// TIA Portal V19 export
FUNCTION_BLOCK "LAF_MemCardDiag"   // FB59, LAD
TITLE = LAF_MemCardDiag / SiemensMemoryCard Diagnose mit ProDiag
AUTHOR : Siemens Digital Industries
FAMILY : LAF
VERSION : 1.2
// Information about the inserted SIMATIC memory card are retrieved, such as  
// * Memory size and assigned memory space of the memory card.  
// * Previously used up portion of the service life (lifetime) and set proportion of the lifetime of the memory card.  
// The data is evaluated in the FB, incl. ProDiag supervisions; it is displayed on the HMI in screen "Settings - PLC & HMI".
// 
// **PLC-Data types**  
// * LAF_typeMemCardDiag  
// * LAF_typeMemCardMessages  
// 
// 
// **WinCC-Screen**  
// 
// ![Image](LAF_MemCardDiag_PrD/en/image2.PNG)
//  
// **Block call example**  
// {.pageWidth}
// ![Image](LAF_MemCardDiag_PrD/en/image10.PNG)
// View in ladder logic (LAD).  
// 
// **Calling interface**  
// The block will be called once only in the cyclic program. The call takes place in the software unit CentralFunctions -> 05_Diagnostic -> [CallDiagnostic](../Functions/CallDiagnostic.htm)  
//   
// 
// **Internally used “Extended instructions / blocks”**  
// GetSMCinfo  
// 
// **Parameters**  
// 
// This block is provided with “pre-defined actual parameters” for structured data types, user constants, system constants etc. Therefor these parameters have to be modified only slightly or not at all, if the symbols of DBs, user constants, and system constants have not been changed.
// Es werden Informationen über die in der CPU gesteckte Memory Card ausgelesen, wie:  
// * Zur Verfügung stehender und benutzter Speicherplatz der Memory Card 
// * Verbrauchter Anteil und Parametrierter Anteil der Lebensdauer der Memory Card 
// 
// Die Daten werden in dem FB ausgewertet incl. ProDiag-Meldungen und auf dem HMI im Bild „SYSTEM_SETTINGS“ und im Bildbaustein „SMC_Diag“ dargestellt.  
// * LSicar_MemCardDiag_PrD:		mit ProDiag-Meldeverfahren 
// * LSicar_MemCardDiag		mit program_Alarm Meldeverfahren 
// 
// **PLC-Datentypen**  
// * LSicar_typeMemCardDiag 
// * LSicar_typeMemCardMessages  
// 
// 
// **WinCC-Faceplate**  
// 
// ![Image](LSicar_MemCardDiag_PrD/de/image1.PNG)
// 
// **WinCC-Bild**  
// 
// ![Image](LSicar_MemCardDiag_PrD/de/image2.PNG)
//  
// **Beispielaufruf**  
// Abbildung in Kontaktplan (KOP), ohne Parameterbeschaltung.  
// 
// **Aufrufschnittstelle**  
// Der Baustein wird einmalig im zyklischen Programm aufgerufen im FC „CallDiagnostic“  
// 
// **Intern verwendete „Erweiterte Anweisungen / Instructions“**  
// GetSMCinfo  
// 
// **Parameter**  
// 
// ![Icon](_Icon/information.PNG)
// 
// Der Baustein ist mit "Vordefinierten Aktualparametern" versehen für Strukturvariablen, Anwender- und Systemkonstanten etc., die dadurch nicht oder nur geringfügig angepasst werden müssen, vorausgesetzt die Symbolischen Namen von DBs, Anwender-/Systemkonstanten etc. wurden nicht geändert. Die Anpassungen sind notwendig beim Index [i], z.B. für den BA-Bereich oder die HMI-/Panelnummer.  
// * Der Index ist vorbesetzt mit dem Wert [0]. Damit wird auf den Index 0 (Dummy) verwiesen. Sofern der Baustein-Parameter nicht benötigt wird, sind keine Anpassungen notwendig, andernfalls muss der Indexwert angepasst werden. 
// oder  
// * Der Index ist vorbesetzt mit [???]. Dies führt dazu, dass der Aktualparameter beim Bausteinaufruf rot markiert wird; um darauf aufmerksam zu machen, dass der Indexwert des Aktualparameters angepasst werden muss!
// stored: Access Published, IsIECCheckEnabled true, MemoryReserve 100, SetENOAutomatically true
   VAR_INPUT
      plantIdentifier { ExternalAccessible := 'False'; ExternalVisible := 'False'; ExternalWritable := 'False'} : WString[#MAX_CHAR];   // Betriebsmittel Kennzeichen. Das Kennzeichen ist auf 24 Zeichen begrenzt und sollte ein Betriebsmittelkennzeichen, gemäß der Schaltpläne enthalten. Der hier angegebene Text dient als Präfix und erscheint im ProDiag-Meldetext in der Meldeanzeige. / Identifier of the device. The identifier is limited to a length of 24 characters and should contain the name of the device according the wiring diagrams. The identifier is displayed as a prefix for the alarm messages..
      textListId { ExternalAccessible := 'False'; ExternalVisible := 'False'; ExternalWritable := 'False'} : Int;   // Text list ID
      firstCycle { ExternalAccessible := 'False'; ExternalVisible := 'False'; ExternalWritable := 'False'} : Bool;   // Variable die den ersten CPU-Zyklus darstellt. Im ersten Zyklus werden alle Informationen einmalig gelesen und dargestellt. / Tag representing the first CPU cycle. All information is read and stored once in the first CPU cycle.
      readInfoMemCard { ExternalAccessible := 'False'; ExternalVisible := 'False'; ExternalWritable := 'False'} : Bool;   // Mit einem Wechsel 0 auf 1 Signal werden ebenso die Informationen einmalig gelesen und dargestellt. Hinweis: Es ist nicht notwendig die Informationen CPU-zyklisch auszulesen. Verwenden Sie daher ein geeignetes Signal um die Zyklusbelastung gering zu halten. / All information is read and stored once if the state of this parameter changes from FALSE to TRUE. Note: it is not necessary to read the information in each cycle of the CPU. Therefor use a suitable signal to keep the cycle load.
      hideAlarmMask { ExternalAccessible := 'False'; ExternalVisible := 'False'; ExternalWritable := 'False'} : Byte;   // Einzelne Störungen unterdrücken. Bei Bedarf können einzelne Meldungen deaktiviert werden, durch Setzen des entsprechenden Bits auf TRUE. Belegung: siehe AlarmWarnInfo / Suppress single alarms. If required single alarms can be deactivated by putting the corresponding bit on TRUE.
   END_VAR
   VAR_OUTPUT
      generalAlarm { ExternalAccessible := 'False'; ExternalVisible := 'False'; ExternalWritable := 'False'} : Bool;   // Sammelbit für Alarm / Collective signal for alarm
      generalWarn { ExternalAccessible := 'False'; ExternalVisible := 'False'; ExternalWritable := 'False'} : Bool;   // Sammelbit für Alarm / Collective signal for warning
      generalInfo { ExternalAccessible := 'False'; ExternalVisible := 'False'; ExternalWritable := 'False'} : Bool;   // Sammelbit für Information / Collective signal for information
   END_VAR
   VAR_IN_OUT
      diagHmi : "LAF_typeMemCardDiag";   // Transfer of the information for display on the HMI. The parameter is predefined and refers to the specified destination. / Übergabe der Informationen zur Anzeige am HMI. Der Para-meter ist vordefiniert und verweist auf angegebenes Ziel
   END_VAR
   VAR
      statMessages { ExternalAccessible := 'False'; ExternalVisible := 'False'; ExternalWritable := 'False'} : "LAF_typeMemCardMessages";   // Störungen/Warnungen/Informationen
      statHideMessages { ExternalAccessible := 'False'; ExternalVisible := 'False'; ExternalWritable := 'False'} : "LAF_typeMemCardMessages";   // Störungen/Warnungen/Informationen unterdrücken / Hide Alarms/Warnings/Information
      statStep { ExternalAccessible := 'False'; ExternalVisible := 'False'; ExternalWritable := 'False'} : Array[0..3] of Bool;   // Startbits für GetSMCinfo, Mode0..3 / Startbits for GetSMCinfo, Mode0..3
      statRisEdgeStep0 { ExternalAccessible := 'False'; ExternalVisible := 'False'; ExternalWritable := 'False'} : Bool;   // Steigende Flanke / Rising edge
      statRisEdgeStep1 { ExternalAccessible := 'False'; ExternalVisible := 'False'; ExternalWritable := 'False'} : Bool;   // Rising edge step0 / Steigende Flanke
      statAlarmNo { ExternalAccessible := 'False'; ExternalVisible := 'False'; ExternalWritable := 'False'} : UInt;   // Alarm Nummer für ProDiag / Alarm Number for ProDiag
      statWarnNo { ExternalAccessible := 'False'; ExternalVisible := 'False'; ExternalWritable := 'False'} : UInt;   // Warn Nummer für ProDiag / Warn Number for ProDiag
      statInfoNo { ExternalAccessible := 'False'; ExternalVisible := 'False'; ExternalWritable := 'False'} : UInt;   // Info Nummer für ProDiag / Info Number for ProDiag
      instGetInfoMode0 { ExternalAccessible := 'False'; ExternalVisible := 'False'; ExternalWritable := 'False'} : GetSMCinfo;   // GetSMCinfo
      instGetInfoMode1 { ExternalAccessible := 'False'; ExternalVisible := 'False'; ExternalWritable := 'False'} : GetSMCinfo;   // GetSMCinfo
      instGetInfoMode2 { ExternalAccessible := 'False'; ExternalVisible := 'False'; ExternalWritable := 'False'} : GetSMCinfo;   // GetSMCinfo
      instGetInfoMode3 { ExternalAccessible := 'False'; ExternalVisible := 'False'; ExternalWritable := 'False'} : GetSMCinfo;   // GetSMCinfo
   END_VAR
   VAR CONSTANT
      MAX_CHAR : DInt := 24;   // Konstante für Zeichenlänge plantidentifier / Constant length plantidentifier
      ERROR_CODE_8080 : Word := 16#8080;   // Konstante Error code 8080 / Constant error code 8080
      ERROR_CODE_8081 : Word := 16#8081;   // Konstante Error code 8081 / Constant error code 8081
      ERROR_CODE_8092 : Word := 16#8092;   // Konstante Error code 8092 / Constant error code 8092
      ERROR_CODE_80C3 : Word := 16#80C3;   // Konstante Error code 80C3 / Constant error code 80C3
   END_VAR
   VAR_TEMP   // added for the SCL form of the ladder/FBD networks
      _w1 : Bool;
      _w2 : Bool;
      _w3 : Bool;
   END_VAR
BEGIN

REGION Network 1: ChangeLog / Änderungshistorie
   // SIEMENS AG / (c)Copyright 2024
   // ------------------------------------------------------------------------------
   // Title:            LAF_MemCardDiag
   // Comment/Function: Information about the inserted SIMATIC memory card are retrieved
   // Library/Family:           Library of Automation Framework
   // Author:               Siemens Digital Industry
   // Tested with:      S7-PLCSIM Advanced 6.0
   // Engineering:     TIA Portal V19
   // Restrictions:      ---
   // Requirements:  ---
   // ------------------------------------------------------------------------------
   // Change log table:
   // Version | Date | Expert in charge | Changes applied
   // -------|---------|-------------|--------------------------------------------
   // 01.02.00 | 30.09.2024 | SIMATIC Systems Support | First released version
   // Die Änderungshistorie wird nur in englischer Editiersprache geführt.
END_REGION

REGION Network 2: Description / Beschreibung
   // **Operation mode Automatic**  
   // The block is not assigned to any operation mode area.  
   // 
   // **AlarmWarnInfo**  
   // Alarms, warnings and information are stored in the PLC alarm text lists of the software unit GlobalData. This messages are used with proDiag and also in the program alarm version of the block.  
   // 
   // | No. | Message                                                                                     |
   // |-----|---------------------------------------------------------------------------------------------|
   // | 1   | Invalid value of the parameter   "Mode"                                                     |
   // | 2   | No SIMATIC memory card inserted                                                             |
   // | 3   | No data available, eg. "GetSMCinfo" is not supported by the   PLC/SMC                       |
   // | 4   | The maximum of simultaneous calls of "GetSMCinfo" instruction   reached                     |
   // | 5   | Configured memory space for warning reached                                                 |
   // | 6   | Configured memory space for alarm reached                                                   |
   // | 7   | Consumed proportion of service life bigger than the configured proportion   of service life |
   // | 8   | S7-PLCSIM active or diagnostic alarm disabled (PLC properties)                              |
   // 
   // ---
   // 
   // #### PLC settings 
   // Set the check box for “Aging of the SIMATIC memory card” in “CPU properties / SIMATIC memory card” and select the threshold value.  
   // ![Image](LAF_MemCardDiag_PrD/en/image5.PNG)
   // 
   // #### Define memory threshold 
   // The thresholds for the alarm and warning of the memory space are defined as default values in the Settings DB.
   // ![Image](LAF_MemCardDiag_PrD/en/image6.PNG)
   // 
   // 
   // 
   // #### PLC Data types  
   // * [LAF_typeMemCardDiag](../Library%20Types/LAF_typeMemCardDiag.htm)  
   // * [LAF_typeMemCardMessages](../Library%20Types/LAF_typeMemCardMessages.htm)  
   // 
   // #### WinCC-Objects 
   // 
   // The memory card area of the setting screen consists of several WinCC objects. There are colored symbols to indicate the status of the SMC.  
   // 
   // ![Image](LAF_MemCardDiag_PrD/en/image8.PNG)  
   // 
   // If the defined threshold for memory space warning or alarm is exceeded, a red sign for alarm or an orange one for warning appears. 
   // Also, a red sign appears, if the lifetime used up is greater than the configured share of the lifetime additionally to the red sign in the setting screen there is a red clock symbol appearing on the memory card picture in the header screen. 
   // The signs are invisible when no alarm or warning is active.  
   // 
   // **WinCC Faceplate**  
   // The faceplate “LAF_MemCardDiag” is stored in the project library. It is shown with a clock symbol, if the configured life time threshold is exceeded.  
   // ![Image](LAF_MemCardDiag_PrD/en/image9.PNG)
   // 
   // 
   // 
   // #### Further information 
   // 
   // #### Update info 
   // 
   // #### Further documentation
   // **Betriebsart Automatik / Hand**  
   // Der Baustein ist keinem Betriebsartenbereich zugeordnet.  
   // 
   // **AlarmWarnInfo**  
   // Alarme, Warnungen und Informationen sind im Statischen Teil in der Struktur „AlarmWarnInfo“ abgebildet.  
   // Der dem Bit %X0…%X7 zugehörige Text der PLC-Meldetextliste erscheint in der ProDiag-Meldung. Durch das Setzen des Bits %X0…%X7 in „hideAlarmMask“ unterdrücken Sie die Meldung.  
   // 
   // ![Image](LSicar_MemCardDiag_PrD/de/image3.PNG)
   //  
   // %X0  
   // %X1  
   // %X2  
   // %X3  
   // %X4  
   // %X5  
   // %X6  
   // %X7  
   // 
   // **PLC-Meldetextliste**  
   // Die PLC-Meldetextliste „SMC_Diag_AlarmWarnInfo_PD“ beinhaltet die Meldetexte wie oben angegeben. Die Texte werden in der ProDiag-Meldung ausgegeben. Sie ist zweisprachig ausgelegt (deutsch, englisch).  
   // Die PLC-Meldetextliste ist in den SICAR-Projekten aufgerufen in „GLOBAL_GENERAL_AlarmTextList“.  
   // Beachten Sie hier ebenso die Mehrsprachigkeit der Einträge.  
   // 
   // ![Image](LSicar_MemCardDiag_PrD/de/image4.PNG)
   //  
   // 
   //  
   // 
   // #### CPU Einstellungen
   // Setzen Sie hierzu das Häkchen „Lebensdauer der SIMATIC Memory Card“ in den CPU-Einstellungen und wählen Sie den Schwellenwert.
   //   
   // ![Image](LSicar_MemCardDiag_PrD/de/image5.PNG)
   //  
   // 
   // #### PLC-Datentypen 
   // Verwendete PLC-Datentypen für den SPS-Programmbaustein und WinCC-Bildbausteine (Faceplates).  
   // 
   // **_typeMemCardDiag**  
   // 
   // ![Image](LSicar_MemCardDiag_PrD/de/image6.PNG)
   // 
   // enthält die Informationen, die in der Visualisierung angezeigt werden  
   // 
   // **„_typeMemCardMessages**  
   // 
   // ![Image](LSicar_MemCardDiag_PrD/de/image7.PNG)
   // 
   // enthält die möglichen Meldungen, die bei der Funktion SMCDiag generiert werden.  
   // 
   // 
   // #### WinCC-Objekte 
   // 
   // **WinCC-Bildbaustein**  
   // Der Bildbaustein befindet sich in der Projekt-Bibliothek unter „Typen“.  
   // Der Bildbaustein ist erstellt aus mehreren einzelnen WinCC-Objekten. Er wird farblich animiert, je nach Zustand.  
   // 
   // ![Image](LSicar_MemCardDiag_PrD/de/image8.PNG)
   // 
   // * Schwarz: Gut-Zustand 
   // * Helles Orange:  1  Parametrierte Speicherkapazität für Warnung erreicht 
   // * Hellrot:  2  Parametrierte Speicherkapazität für Alarm erreicht 
   // * Kleines rotes Kreuz unten rechts im Bildbaustein:  
   // * Keine SMC-Karte gesteckt (nur bei S7-1200) 
   // * Rotes Uhrsymbol unten links im Bildbaustein: 3 Verbrauchter Anteil der Lebensdauer ist größer wie der parametrierte Anteil der Lebensdauer.
   // 
   // Schnittstelle des Bildbausteins:  
   // Für die Schnittstelle des Bildbausteins ist die HMI-Variable „GlobalInterface_SMCDiagHMI_AlarmWarnInfo“ verwendet.  
   // 
   // **WinCC-Bild**  
   // Die einzelnen HMI-Objekte für die SMC-Diagnose sind im Bild „SYSTEM_SETTINGS“ enthalten.  
   // 
   // ![Image](LSicar_MemCardDiag_PrD/de/image9.PNG)  
   // 
   // 
   // ####  Weitere Hinweise
   // 
   // #### Updateinfo 
   // 
   // #### Weitere Dokumente
END_REGION

REGION Network 3: General / preparations / Allgemein/Vorbereitungen
   // Initialization of the step flags / Initialisieren der Schrittvariablen
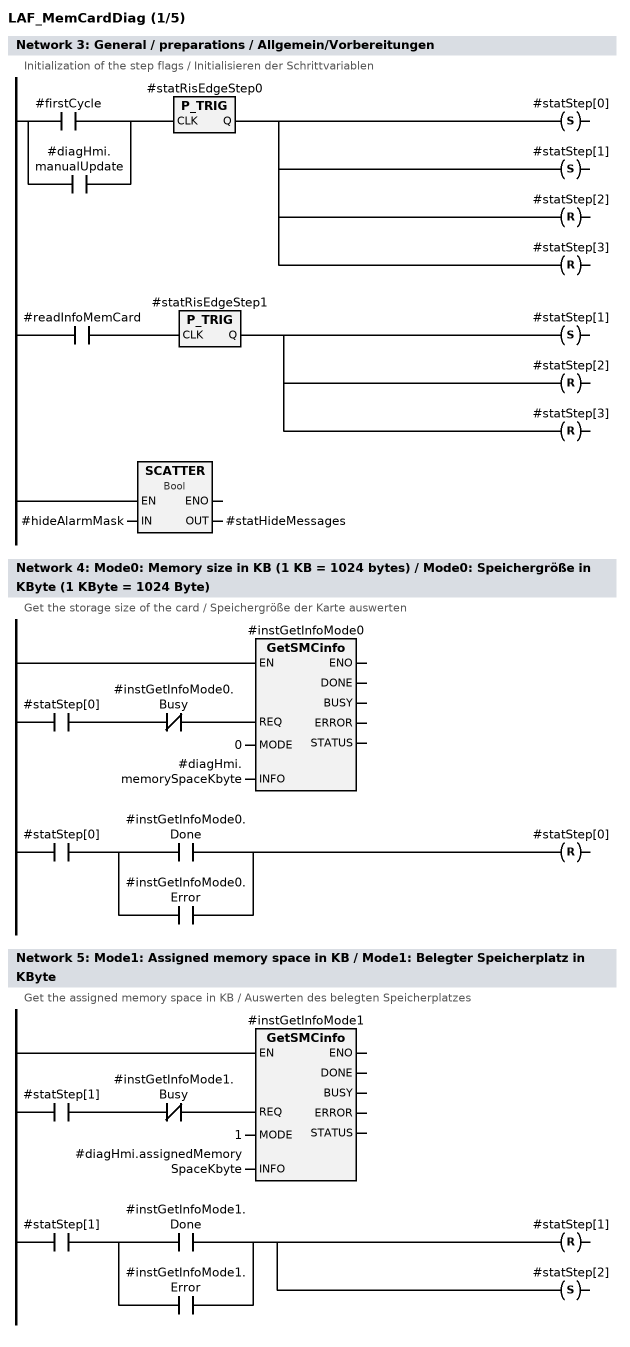
   RUNG wire#powerrail
      Contact( #firstCycle )
      wire#w1
      P_Trig( #statRisEdgeStep0 )
      wire#w2
      S_Coil( #statStep[0] )
   END_RUNG
   RUNG wire#powerrail
      Contact( #diagHmi.manualUpdate )
   END_RUNG wire#w1
   RUNG wire#w2
      S_Coil( #statStep[1] )
   END_RUNG
   RUNG wire#w2
      R_Coil( #statStep[2] )
   END_RUNG
   RUNG wire#w2
      R_Coil( #statStep[3] )
   END_RUNG
   RUNG wire#powerrail
      Contact( #readInfoMemCard )
      P_Trig( #statRisEdgeStep1 )
      wire#w3
      S_Coil( #statStep[1] )
   END_RUNG
   RUNG wire#w3
      R_Coil( #statStep[2] )
   END_RUNG
   RUNG wire#w3
      R_Coil( #statStep[3] )
   END_RUNG
   RUNG wire#powerrail
      { S7_Templates := "[dest_type := Bool, src_type := Byte]" } SCATTER(IN := #hideAlarmMask, OUT => #statHideMessages)
   END_RUNG
   // the same network as SCL:
   #_w1 := #firstCycle OR #diagHmi.manualUpdate;
   #_w2 := #_w1 AND NOT #statRisEdgeStep0;   // rising edge
   #statRisEdgeStep0 := #_w1;
   IF #_w2 THEN
       #statStep[0] := TRUE;
       #statStep[1] := TRUE;
       #statStep[2] := FALSE;
       #statStep[3] := FALSE;
   END_IF;
   #_w3 := #readInfoMemCard AND NOT #statRisEdgeStep1;   // rising edge
   #statRisEdgeStep1 := #readInfoMemCard;
   IF #_w3 THEN
       #statStep[1] := TRUE;
       #statStep[2] := FALSE;
       #statStep[3] := FALSE;
   END_IF;
   SCATTER(IN := #hideAlarmMask, OUT => #statHideMessages);
END_REGION

REGION Network 4: Mode0: Memory size in KB (1 KB = 1024 bytes) / Mode0: Speichergröße in KByte (1 KByte = 1024 Byte)
   // Get the storage size of the card / Speichergröße der Karte auswerten
   RUNG wire#powerrail
      #instGetInfoMode0.GetSMCinfo(REQ := wire#w1, Mode := 0, Info := #diagHmi.memorySpaceKbyte, Done =>, Busy =>, Error =>, Status =>)
   END_RUNG
   RUNG wire#powerrail
      Contact( #statStep[0] )
      I_Contact( #instGetInfoMode0.Busy )
   END_RUNG wire#w1
   RUNG wire#powerrail
      Contact( #statStep[0] )
      wire#w2
      Contact( #instGetInfoMode0.Done )
      wire#w3
      R_Coil( #statStep[0] )
   END_RUNG
   RUNG wire#w2
      Contact( #instGetInfoMode0.Error )
   END_RUNG wire#w3
   // the same network as SCL:
   #instGetInfoMode0(REQ := #statStep[0] AND NOT #instGetInfoMode0.Busy,   // GetSMCinfo
                     Mode := 0,
                     Info := #diagHmi.memorySpaceKbyte);
   IF #statStep[0] AND (#instGetInfoMode0.Done OR #instGetInfoMode0.Error) THEN
       #statStep[0] := FALSE;
   END_IF;
END_REGION

REGION Network 5: Mode1: Assigned memory space in KB / Mode1: Belegter Speicherplatz in KByte
   // Get the assigned memory space in KB / Auswerten des belegten Speicherplatzes
   RUNG wire#powerrail
      #instGetInfoMode1.GetSMCinfo(REQ := wire#w1, Mode := 1, Info := #diagHmi.assignedMemorySpaceKbyte, Done =>, Busy =>, Error =>, Status =>)
   END_RUNG
   RUNG wire#powerrail
      Contact( #statStep[1] )
      I_Contact( #instGetInfoMode1.Busy )
   END_RUNG wire#w1
   RUNG wire#powerrail
      Contact( #statStep[1] )
      wire#w2
      Contact( #instGetInfoMode1.Done )
      wire#w3
      R_Coil( #statStep[1] )
   END_RUNG
   RUNG wire#w2
      Contact( #instGetInfoMode1.Error )
   END_RUNG wire#w3
   RUNG wire#w3
      S_Coil( #statStep[2] )
   END_RUNG
   // the same network as SCL:
   #instGetInfoMode1(REQ := #statStep[1] AND NOT #instGetInfoMode1.Busy,   // GetSMCinfo
                     Mode := 1,
                     Info := #diagHmi.assignedMemorySpaceKbyte);
   #_w1 := #statStep[1] AND (#instGetInfoMode1.Done OR #instGetInfoMode1.Error);
   IF #_w1 THEN
       #statStep[1] := FALSE;
       #statStep[2] := TRUE;
   END_IF;
END_REGION

REGION Network 6: Mode2: Maintenance information consumed lifetime / Mode2: Wartungsinformation verbrauchte Lebenszeit
   // Previously used up portion of the service life in % / Bisher verbrauchter Anteil der Lebensdauer in %
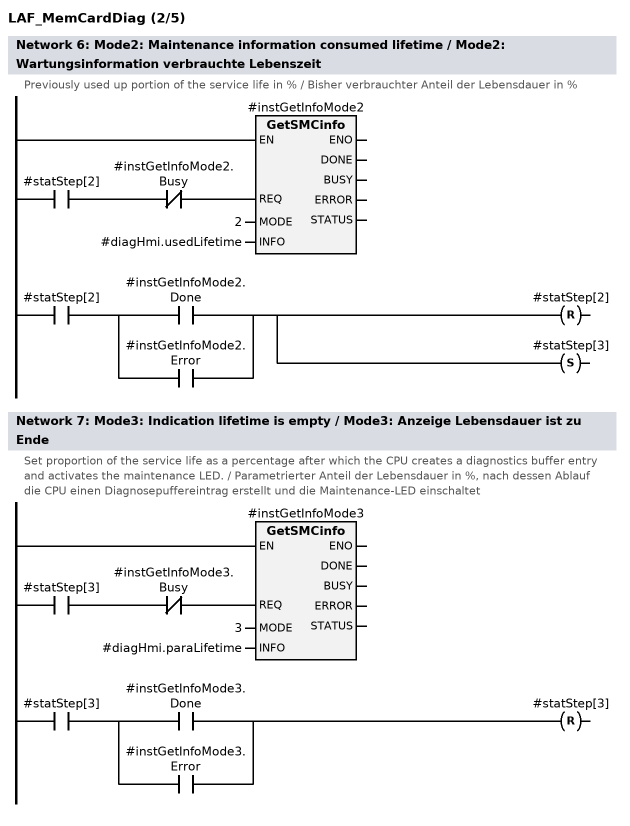
   RUNG wire#powerrail
      #instGetInfoMode2.GetSMCinfo(REQ := wire#w1, Mode := 2, Info := #diagHmi.usedLifetime, Done =>, Busy =>, Error =>, Status =>)
   END_RUNG
   RUNG wire#powerrail
      Contact( #statStep[2] )
      I_Contact( #instGetInfoMode2.Busy )
   END_RUNG wire#w1
   RUNG wire#powerrail
      Contact( #statStep[2] )
      wire#w2
      Contact( #instGetInfoMode2.Done )
      wire#w3
      R_Coil( #statStep[2] )
   END_RUNG
   RUNG wire#w2
      Contact( #instGetInfoMode2.Error )
   END_RUNG wire#w3
   RUNG wire#w3
      S_Coil( #statStep[3] )
   END_RUNG
   // the same network as SCL:
   #instGetInfoMode2(REQ := #statStep[2] AND NOT #instGetInfoMode2.Busy,   // GetSMCinfo
                     Mode := 2,
                     Info := #diagHmi.usedLifetime);
   #_w1 := #statStep[2] AND (#instGetInfoMode2.Done OR #instGetInfoMode2.Error);
   IF #_w1 THEN
       #statStep[2] := FALSE;
       #statStep[3] := TRUE;
   END_IF;
END_REGION

REGION Network 7: Mode3: Indication lifetime is empty / Mode3: Anzeige Lebensdauer ist zu Ende
   // Set proportion of the service life as a percentage after which the CPU creates a diagnostics buffer entry and activates the maintenance LED. / Parametrierter Anteil der Lebensdauer in %, nach dessen Ablauf die CPU einen Diagnosepuffereintrag erstellt und die Maintenance-LED einschaltet
   RUNG wire#powerrail
      #instGetInfoMode3.GetSMCinfo(REQ := wire#w1, Mode := 3, Info := #diagHmi.paraLifetime, Done =>, Busy =>, Error =>, Status =>)
   END_RUNG
   RUNG wire#powerrail
      Contact( #statStep[3] )
      I_Contact( #instGetInfoMode3.Busy )
   END_RUNG wire#w1
   RUNG wire#powerrail
      Contact( #statStep[3] )
      wire#w2
      Contact( #instGetInfoMode3.Done )
      wire#w3
      R_Coil( #statStep[3] )
   END_RUNG
   RUNG wire#w2
      Contact( #instGetInfoMode3.Error )
   END_RUNG wire#w3
   // the same network as SCL:
   #instGetInfoMode3(REQ := #statStep[3] AND NOT #instGetInfoMode3.Busy,   // GetSMCinfo
                     Mode := 3,
                     Info := #diagHmi.paraLifetime);
   IF #statStep[3] AND (#instGetInfoMode3.Done OR #instGetInfoMode3.Error) THEN
       #statStep[3] := FALSE;
   END_IF;
END_REGION

REGION Network 8: Create errors / Erstellen von Fehlermeldungen
   // Create Alarms/Warnings from Errorcode / Alarme/Warnungen bilden aus Fehlercode
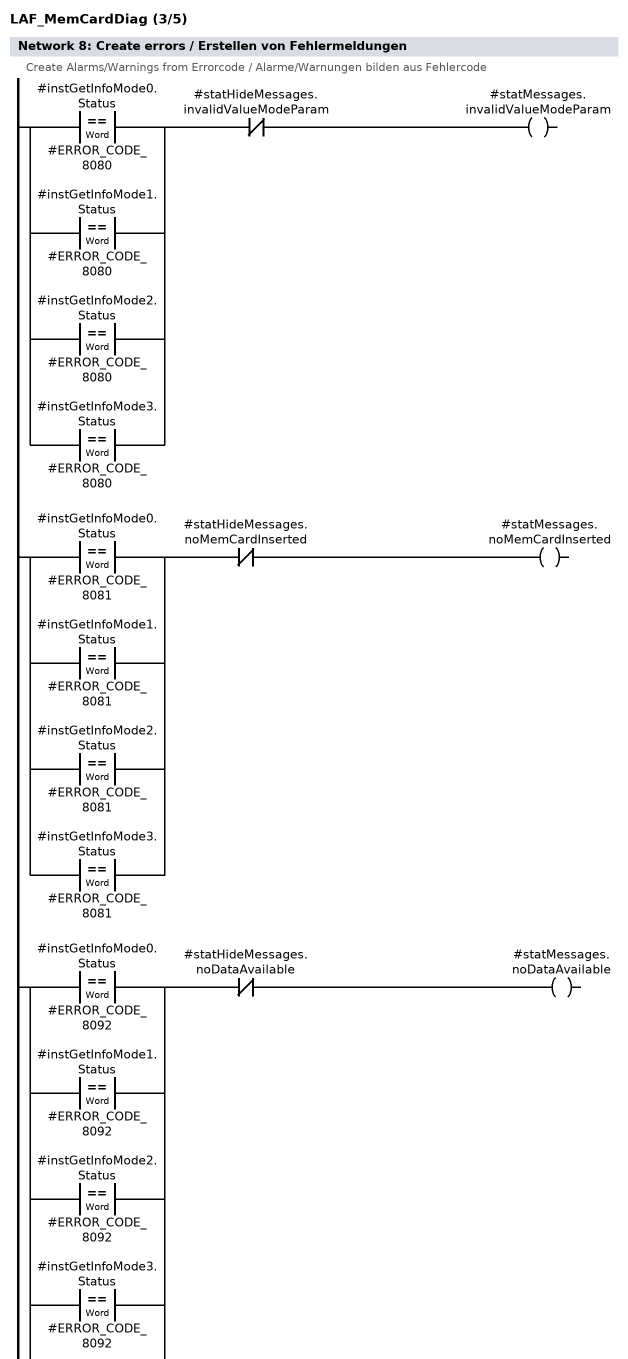
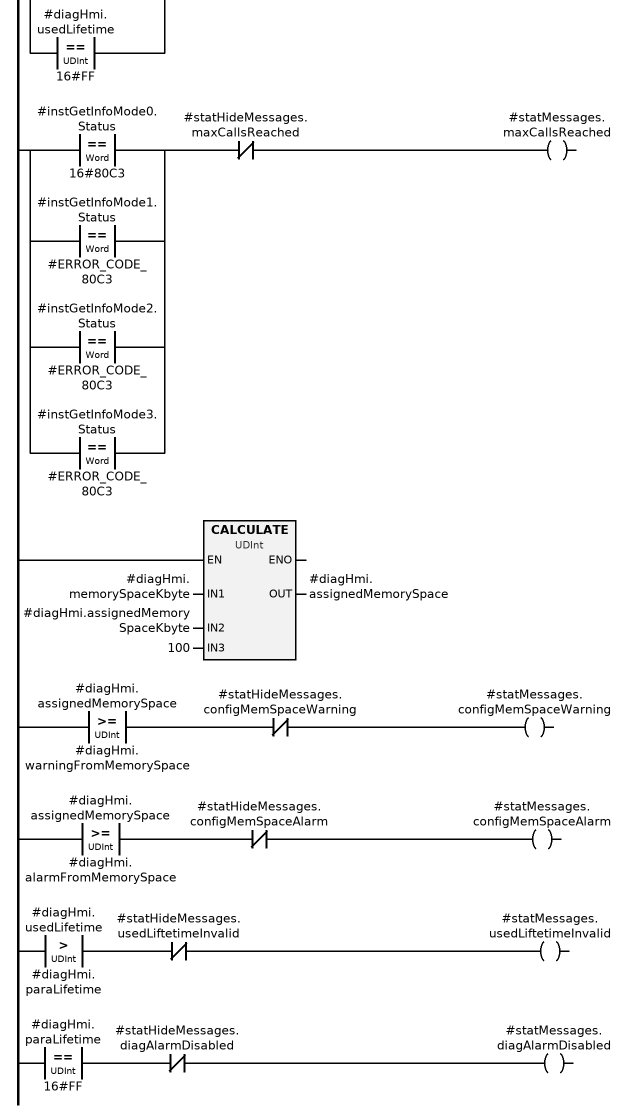
   RUNG wire#powerrail
      { S7_Templates := "SrcType := Word" } EQ_Contact(in1 := #instGetInfoMode0.Status, in2 := #ERROR_CODE_8080)
      wire#w1
      I_Contact( #statHideMessages.invalidValueModeParam )
      Coil( #statMessages.invalidValueModeParam )
   END_RUNG
   RUNG wire#powerrail
      { S7_Templates := "SrcType := Word" } EQ_Contact(in1 := #instGetInfoMode1.Status, in2 := #ERROR_CODE_8080)
   END_RUNG wire#w1
   RUNG wire#powerrail
      { S7_Templates := "SrcType := Word" } EQ_Contact(in1 := #instGetInfoMode2.Status, in2 := #ERROR_CODE_8080)
   END_RUNG wire#w1
   RUNG wire#powerrail
      { S7_Templates := "SrcType := Word" } EQ_Contact(in1 := #instGetInfoMode3.Status, in2 := #ERROR_CODE_8080)
   END_RUNG wire#w1
   RUNG wire#powerrail
      { S7_Templates := "SrcType := Word" } EQ_Contact(in1 := #instGetInfoMode0.Status, in2 := #ERROR_CODE_8081)
      wire#w2
      I_Contact( #statHideMessages.noMemCardInserted )
      Coil( #statMessages.noMemCardInserted )
   END_RUNG
   RUNG wire#powerrail
      { S7_Templates := "SrcType := Word" } EQ_Contact(in1 := #instGetInfoMode1.Status, in2 := #ERROR_CODE_8081)
   END_RUNG wire#w2
   RUNG wire#powerrail
      { S7_Templates := "SrcType := Word" } EQ_Contact(in1 := #instGetInfoMode2.Status, in2 := #ERROR_CODE_8081)
   END_RUNG wire#w2
   RUNG wire#powerrail
      { S7_Templates := "SrcType := Word" } EQ_Contact(in1 := #instGetInfoMode3.Status, in2 := #ERROR_CODE_8081)
   END_RUNG wire#w2
   RUNG wire#powerrail
      { S7_Templates := "SrcType := Word" } EQ_Contact(in1 := #instGetInfoMode0.Status, in2 := #ERROR_CODE_8092)
      wire#w3
      I_Contact( #statHideMessages.noDataAvailable )
      Coil( #statMessages.noDataAvailable )
   END_RUNG
   RUNG wire#powerrail
      { S7_Templates := "SrcType := Word" } EQ_Contact(in1 := #instGetInfoMode1.Status, in2 := #ERROR_CODE_8092)
   END_RUNG wire#w3
   RUNG wire#powerrail
      { S7_Templates := "SrcType := Word" } EQ_Contact(in1 := #instGetInfoMode2.Status, in2 := #ERROR_CODE_8092)
   END_RUNG wire#w3
   RUNG wire#powerrail
      { S7_Templates := "SrcType := Word" } EQ_Contact(in1 := #instGetInfoMode3.Status, in2 := #ERROR_CODE_8092)
   END_RUNG wire#w3
   RUNG wire#powerrail
      { S7_Templates := "SrcType := UDInt" } EQ_Contact(in1 := #diagHmi.usedLifetime, in2 := 16#FF)
   END_RUNG wire#w3
   RUNG wire#powerrail
      { S7_Templates := "SrcType := Word" } EQ_Contact(in1 := #instGetInfoMode0.Status, in2 := 16#80C3)
      wire#w4
      I_Contact( #statHideMessages.maxCallsReached )
      Coil( #statMessages.maxCallsReached )
   END_RUNG
   RUNG wire#powerrail
      { S7_Templates := "SrcType := Word" } EQ_Contact(in1 := #instGetInfoMode1.Status, in2 := #ERROR_CODE_80C3)
   END_RUNG wire#w4
   RUNG wire#powerrail
      { S7_Templates := "SrcType := Word" } EQ_Contact(in1 := #instGetInfoMode2.Status, in2 := #ERROR_CODE_80C3)
   END_RUNG wire#w4
   RUNG wire#powerrail
      { S7_Templates := "SrcType := Word" } EQ_Contact(in1 := #instGetInfoMode3.Status, in2 := #ERROR_CODE_80C3)
   END_RUNG wire#w4
   RUNG wire#powerrail
      { S7_Templates := "SrcType := UDInt"; S7_Expression := "(IN2 * IN3) / IN1" } Calculate(in1 := #diagHmi.memorySpaceKbyte, in2 := #diagHmi.assignedMemorySpaceKbyte, in3 := 100, out => #diagHmi.assignedMemorySpace)
   END_RUNG
   RUNG wire#powerrail
      { S7_Templates := "SrcType := UDInt" } GE_Contact(in1 := #diagHmi.assignedMemorySpace, in2 := #diagHmi.warningFromMemorySpace)
      I_Contact( #statHideMessages.configMemSpaceWarning )
      Coil( #statMessages.configMemSpaceWarning )
   END_RUNG
   RUNG wire#powerrail
      { S7_Templates := "SrcType := UDInt" } GE_Contact(in1 := #diagHmi.assignedMemorySpace, in2 := #diagHmi.alarmFromMemorySpace)
      I_Contact( #statHideMessages.configMemSpaceAlarm )
      Coil( #statMessages.configMemSpaceAlarm )
   END_RUNG
   RUNG wire#powerrail
      { S7_Templates := "SrcType := UDInt" } GT_Contact(in1 := #diagHmi.usedLifetime, in2 := #diagHmi.paraLifetime)
      I_Contact( #statHideMessages.usedLiftetimeInvalid )
      Coil( #statMessages.usedLiftetimeInvalid )
   END_RUNG
   RUNG wire#powerrail
      { S7_Templates := "SrcType := UDInt" } EQ_Contact(in1 := #diagHmi.paraLifetime, in2 := 16#FF)
      I_Contact( #statHideMessages.diagAlarmDisabled )
      Coil( #statMessages.diagAlarmDisabled )
   END_RUNG
   // the same network as SCL:
   #statMessages.invalidValueModeParam := ((#instGetInfoMode0.Status = #ERROR_CODE_8080) OR (#instGetInfoMode1.Status = #ERROR_CODE_8080) OR (#instGetInfoMode2.Status = #ERROR_CODE_8080) OR (#instGetInfoMode3.Status = #ERROR_CODE_8080)) AND NOT #statHideMessages.invalidValueModeParam;
   #statMessages.noMemCardInserted := ((#instGetInfoMode0.Status = #ERROR_CODE_8081) OR (#instGetInfoMode1.Status = #ERROR_CODE_8081) OR (#instGetInfoMode2.Status = #ERROR_CODE_8081) OR (#instGetInfoMode3.Status = #ERROR_CODE_8081)) AND NOT #statHideMessages.noMemCardInserted;
   #statMessages.noDataAvailable := ((#instGetInfoMode0.Status = #ERROR_CODE_8092) OR (#instGetInfoMode1.Status = #ERROR_CODE_8092) OR (#instGetInfoMode2.Status = #ERROR_CODE_8092) OR (#instGetInfoMode3.Status = #ERROR_CODE_8092) OR (#diagHmi.usedLifetime = 16#FF)) AND NOT #statHideMessages.noDataAvailable;
   #statMessages.maxCallsReached := ((#instGetInfoMode0.Status = 16#80C3) OR (#instGetInfoMode1.Status = #ERROR_CODE_80C3) OR (#instGetInfoMode2.Status = #ERROR_CODE_80C3) OR (#instGetInfoMode3.Status = #ERROR_CODE_80C3)) AND NOT #statHideMessages.maxCallsReached;
   #diagHmi.assignedMemorySpace := (#diagHmi.assignedMemorySpaceKbyte * 100) / #diagHmi.memorySpaceKbyte;
   #statMessages.configMemSpaceWarning := (#diagHmi.assignedMemorySpace >= #diagHmi.warningFromMemorySpace) AND NOT #statHideMessages.configMemSpaceWarning;
   #statMessages.configMemSpaceAlarm := (#diagHmi.assignedMemorySpace >= #diagHmi.alarmFromMemorySpace) AND NOT #statHideMessages.configMemSpaceAlarm;
   #statMessages.usedLiftetimeInvalid := (#diagHmi.usedLifetime > #diagHmi.paraLifetime) AND NOT #statHideMessages.usedLiftetimeInvalid;
   #statMessages.diagAlarmDisabled := (#diagHmi.paraLifetime = 16#FF) AND NOT #statHideMessages.diagAlarmDisabled;
END_REGION

REGION Network 9: General Alarm/-Warning/-Information / Sammelstörung/-warnung/-information
   // Evaluate alarms, warnings and informations / Auswerten von Alarmen, Warnungen und Informationen
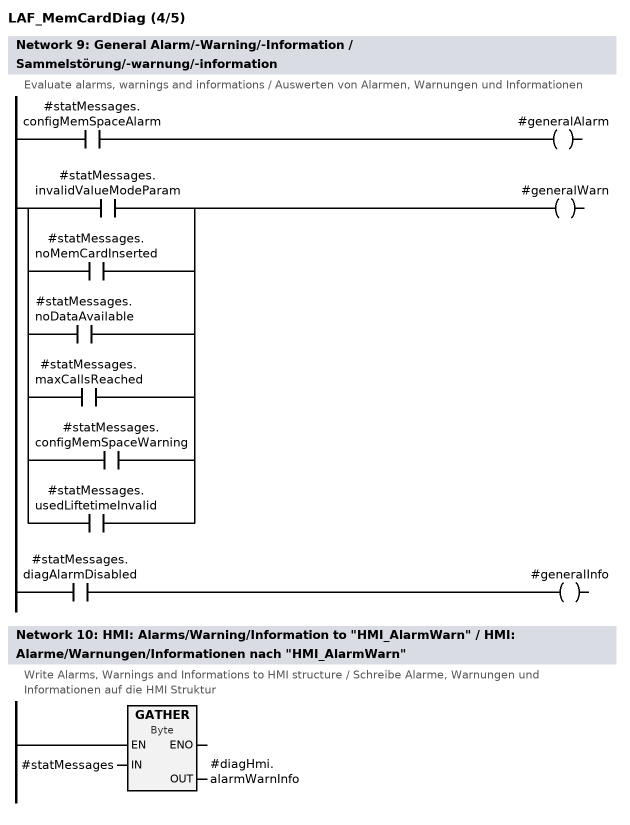
   RUNG wire#powerrail
      Contact( #statMessages.configMemSpaceAlarm )
      Coil( #generalAlarm )
   END_RUNG
   RUNG wire#powerrail
      Contact( #statMessages.invalidValueModeParam )
      wire#w1
      Coil( #generalWarn )
   END_RUNG
   RUNG wire#powerrail
      Contact( #statMessages.noMemCardInserted )
   END_RUNG wire#w1
   RUNG wire#powerrail
      Contact( #statMessages.noDataAvailable )
   END_RUNG wire#w1
   RUNG wire#powerrail
      Contact( #statMessages.maxCallsReached )
   END_RUNG wire#w1
   RUNG wire#powerrail
      Contact( #statMessages.configMemSpaceWarning )
   END_RUNG wire#w1
   RUNG wire#powerrail
      Contact( #statMessages.usedLiftetimeInvalid )
   END_RUNG wire#w1
   RUNG wire#powerrail
      Contact( #statMessages.diagAlarmDisabled )
      Coil( #generalInfo )
   END_RUNG
   // the same network as SCL:
   #generalAlarm := #statMessages.configMemSpaceAlarm;
   #generalWarn := #statMessages.invalidValueModeParam OR #statMessages.noMemCardInserted OR #statMessages.noDataAvailable OR #statMessages.maxCallsReached OR #statMessages.configMemSpaceWarning OR #statMessages.usedLiftetimeInvalid;
   #generalInfo := #statMessages.diagAlarmDisabled;
END_REGION

REGION Network 10: HMI: Alarms/Warning/Information to "HMI_AlarmWarn" / HMI: Alarme/Warnungen/Informationen nach "HMI_AlarmWarn"
   // Write Alarms, Warnings and Informations to HMI structure / Schreibe Alarme, Warnungen und Informationen auf die HMI Struktur
   RUNG wire#powerrail
      { S7_Templates := "[dest_type := Byte, src_type := Bool]" } GATHER(IN := #statMessages, OUT => #diagHmi.alarmWarnInfo)
   END_RUNG
   // the same network as SCL:
   GATHER(IN := #statMessages, OUT => #diagHmi.alarmWarnInfo);
END_REGION

REGION Network 11: HMI: Assignment PLC alarm text list / HMI: Zuweisungen PLC -Meldetextlisten
   // Assign the alarms, warnings and informations to ProDiag / Zuweisen der Alarme, Warnungen und Informationen an ProDiag
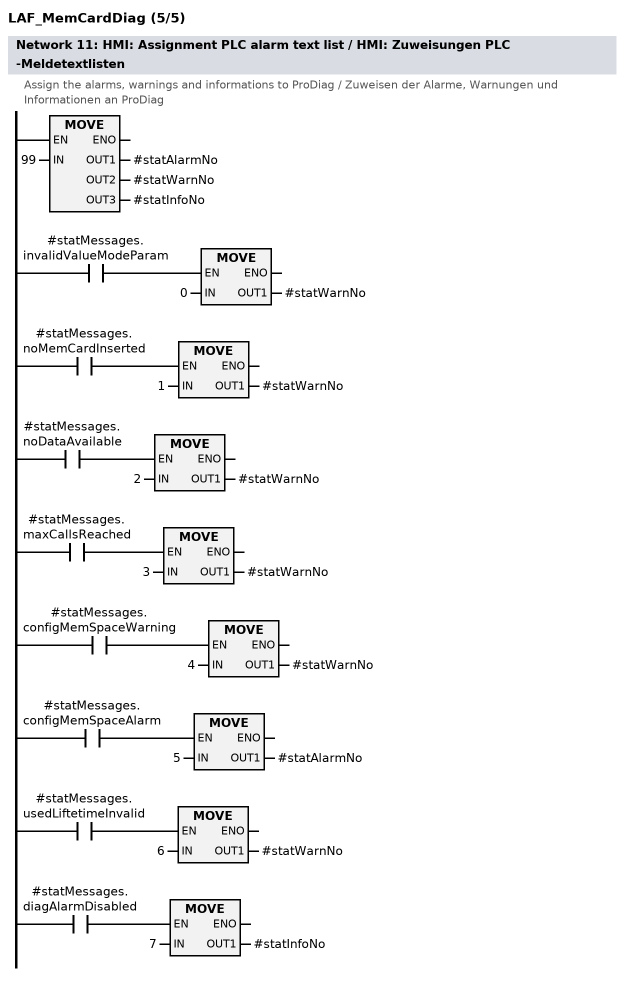
   RUNG wire#powerrail
      Move(in := 99, out1 => #statAlarmNo, out2 => #statWarnNo, out3 => #statInfoNo)
   END_RUNG
   RUNG wire#powerrail
      Contact( #statMessages.invalidValueModeParam )
      Move(in := 0, out1 => #statWarnNo)
   END_RUNG
   RUNG wire#powerrail
      Contact( #statMessages.noMemCardInserted )
      Move(in := 1, out1 => #statWarnNo)
   END_RUNG
   RUNG wire#powerrail
      Contact( #statMessages.noDataAvailable )
      Move(in := 2, out1 => #statWarnNo)
   END_RUNG
   RUNG wire#powerrail
      Contact( #statMessages.maxCallsReached )
      Move(in := 3, out1 => #statWarnNo)
   END_RUNG
   RUNG wire#powerrail
      Contact( #statMessages.configMemSpaceWarning )
      Move(in := 4, out1 => #statWarnNo)
   END_RUNG
   RUNG wire#powerrail
      Contact( #statMessages.configMemSpaceAlarm )
      Move(in := 5, out1 => #statAlarmNo)
   END_RUNG
   RUNG wire#powerrail
      Contact( #statMessages.usedLiftetimeInvalid )
      Move(in := 6, out1 => #statWarnNo)
   END_RUNG
   RUNG wire#powerrail
      Contact( #statMessages.diagAlarmDisabled )
      Move(in := 7, out1 => #statInfoNo)
   END_RUNG
   // the same network as SCL:
   #statAlarmNo := 99;
   #statWarnNo := 99;
   #statInfoNo := 99;
   IF #statMessages.invalidValueModeParam THEN #statWarnNo := 0; END_IF;
   IF #statMessages.noMemCardInserted THEN #statWarnNo := 1; END_IF;
   IF #statMessages.noDataAvailable THEN #statWarnNo := 2; END_IF;
   IF #statMessages.maxCallsReached THEN #statWarnNo := 3; END_IF;
   IF #statMessages.configMemSpaceWarning THEN #statWarnNo := 4; END_IF;
   IF #statMessages.configMemSpaceAlarm THEN #statAlarmNo := 5; END_IF;
   IF #statMessages.usedLiftetimeInvalid THEN #statWarnNo := 6; END_IF;
   IF #statMessages.diagAlarmDisabled THEN #statInfoNo := 7; END_IF;
END_REGION
END_FUNCTION_BLOCK
